FUNCTION_BLOCK FB_BufferStorage
VAR_INPUT
END_VAR
VAR_OUTPUT
	{attribute 'OPC.UA.DA' := '1'}
	localState : ST_BufferStorageState;
END_VAR
VAR
	//sensors
	UpperBufferTemperature : AutomationBaseClasses.FB_TemperatureSensor;
	LowerBufferTemperature : AutomationBaseClasses.FB_TemperatureSensor;
	
	WMZ198 : FB_MollineC3HeatCounter;
	
END_VAR

UpperBufferTemperature();
UpperBufferTemperature.GetState_AI();

LowerBufferTemperature();
LowerBufferTemperature.GetState_AI();

WMZ198(aHeatCounterTelegramm := MBus.Telegramm_WMZ_198);

SetState();

METHOD PROTECTED SetState : BOOL
VAR_INPUT
END_VAR
localState.fUpperTemperature := UpperBufferTemperature.fTemperature;
localState.fLowerTemperature := LowerBufferTemperature.fTemperature;
END_METHOD

END_FUNCTION_BLOCK

(* stored: Version 1.1.0.1, ProductVersion 3.1.4024.6
   POU FB_BufferStorage: Id {bf777c77-d307-4b47-89a9-81af89ea1321}, SpecialFunc None
   Method SetState: Id {b0e6a4ac-cf86-421f-bee7-f1494bba2b38} *)
